// TIA Portal V16 export
// export: Created 2021-03-05T14:22:11.9281466Z, ExportSetting WithDefaults, DisplayName Totally Integrated Automation Portal, DisplayVersion V16, DisplayName TIA Portal Version Control Interface, DisplayVersion V16, DisplayName TIA Portal Openness, DisplayVersion V16, DisplayName SINAMICS Startdrive Advanced, DisplayVersion V16, DisplayName SINAMICS Startdrive G130, G150, S120, S150, SINAMICS MV, S210, DisplayVersion V16, DisplayName SINAMICS Startdrive G110M, G120, G120C, G120D, G120P, DisplayVersion V16, DisplayName STEP 7 Professional, DisplayVersion V16, DisplayName STEP 7 Safety, DisplayVersion V16, DisplayName WinCC Professional, DisplayVersion V16
FUNCTION_BLOCK "fbRoom"   // FB4, LAD
{ S7_Optimized_Access := 'TRUE' }
VERSION : 0.1
// stored: AutoNumber true, IsIECCheckEnabled false, IsRetainMemResEnabled false, MemoryReserve 100, SetENOAutomatically false, UDAEnableTagReadback false
   VAR_INPUT
      arrAI { ExternalAccessible := 'False'; ExternalVisible := 'False'; ExternalWritable := 'False'} : Array[1.."NUM_AI_ROOM"] of Int;
      AI AT arrAI : "udtRoomAI";
   END_VAR
   VAR RETAIN
      Config { ExternalVisible := 'False'; ExternalWritable := 'False'} : Struct
         iNumRacks { ExternalVisible := 'False'; ExternalWritable := 'False'} : Int := 4;
      END_STRUCT;
   END_VAR
   VAR
      Rack { S7_SetPoint := 'True'} : Array[1.."MAX_RACKS_PER_ROOM"] of "fbRack";
      HVAC { S7_SetPoint := 'True'} : "fbRoomHVAC";
   END_VAR
   VAR_TEMP
      i : Int;
      k : Int;
   END_VAR
BEGIN

REGION Network 1 (SCL)
   FOR #i := 1 TO #Config.iNumRacks DO
       #Rack[#i](arrAI := #Rack[#i].arrAI);
   END_FOR;
END_REGION

REGION Network 2 (SCL): HVAC

   #HVAC();
END_REGION
END_FUNCTION_BLOCK
